(* PLC project OOP_Curso, Beckhoff Automation GmbH TwinCAT PLC Control 3.5.13.21 *)
(* stored: creationDateTime 2023-04-24T11:18:57.3670637, modificationDateTime 2023-04-24T11:18:57.3670637 *)

PROGRAM _12_Concepto_Keyword_Abstract
VAR
// 	fbLoadCell:REFERENCE TO AbstractLoadCell;
	
	ConcreteCSVLogger:ConcreteCSVLogger;
    ConcreteAdsLogger:ConcreteADSLogger;
    AbstractLogger:POINTER TO AbstractLogger;
    LogNow:BOOL;
    Process1:INT;
    Process2:INT;
END_VAR

            (*
Concepto ABSTRACTO
La palabra clave ABSTRACT está disponible para bloques de funciones, métodos y propiedades. Permite la implementación de un proyecto PLC con niveles de abstracción.
La abstracción es un concepto clave de la programación orientada a objetos. Los diferentes niveles de abstracción contienen aspectos de implementación generales o específicos.

CONCEPTO ABSTRACTO 1:	
Disponible en TC3.1 Build 4024

Aplicación de la abstracción
Es útil implementar funciones básicas o puntos en común de diferentes clases en una clase básica abstracta. Se implementan aspectos específicos en subclases no abstractas.
El principio es similar al uso de una interfaz. Las interfaces corresponden a clases puramente abstractas que contienen sólo métodos y propiedades abstractas.
Una clase abstracta también puede contener métodos y propiedades no abstractos.

Reglas para el uso de la palabra clave ABSTRACT
Los bloques de funciones abstractas no se pueden instanciar.
Los bloques de funciones abstractas pueden contener métodos y propiedades abstractos y no abstractos.
Los métodos abstractos o las propiedades no contienen ninguna implementación (solo la declaración).
Si un bloque de funciones contiene un método o propiedad abstracta, debe ser abstracta.
Los bloques de funciones abstractas deben extenderse para poder implementar los métodos o propiedades abstractas.
Por lo tanto: Un FB derivado debe implementar los métodos / propiedades de su FB básico o también debe definirse como abstracto.
Muestra
Clase básica abstracta:

FUNCTION_BLOCK ABSTRACT FB_System_Base
Los puntos en común de todos los módulos del sistema se implementan en esta clase básica abstracta. Contiene la propiedad no abstracta "nSystemID" y el método abstracto "Execute" para esto:

PROPERTY nSystemID : UINT
METHOD ABSTRACT Execute
mientras que la implementación de "nSystemID" es la misma para todos los sistemas, la implementación del método "Execute" difiere para los sistemas individuales.

Subclase no abstracta:

FUNCTION_BLOCK FB_StackSystem EXTENDS FB_System_Base
Las clases no abstractas que se derivan de la clase básica se implementan para los sistemas específicos. Esta subclase representa una pila. Dado que no es abstracto, debe implementar el método "Execute" que define la ejecución específica de la pila:

METHOD Execute

*)

// Process 1 assigns a logger and starts task 2.
CASE Process1 OF
    0: IF LogNow THEN
            LogNow:=FALSE;
            AbstractLogger:= ADR(ConcreteAdsLogger);
            Process2 :=1;
            Process1:=Process1+1;               
        END_IF
     
    1: IF Process2 = 0 THEN
            AbstractLogger:= ADR(ConcreteCSVLogger);
            Process2:=1;
            Process1:=Process1+1;   
       END_IF
        
     2:IF Process2 = 0 THEN
            AbstractLogger:= ADR(ConcreteAdsLogger);
            Process2:=1;
            Process1:=Process1+1;   
       END_IF
        
      3: IF Process2 = 0 THEN
            AbstractLogger:= ADR(ConcreteCSVLogger);
            Process2:=1;
            Process1:=Process1+1;   
       END_IF
        
      4:IF Process2 = 0 THEN
            Process1:=0;    
       END_IF
END_CASE
 
//Process 2 does its task indepently of the assigned type of logger. 
CASE process2 OF
    1: AbstractLogger^.LogMessage(CONCAT('Important message ',INT_TO_STRING(Process1)));
       process2:=process2+1;                
         
    2: AbstractLogger^();
       IF NOT AbstractLogger^.Busy THEN
            process2:=0;    
       END_IF
END_CASE
          
END_PROGRAM

FUNCTION_BLOCK ABSTRACT AbstractLoadCell
VAR_INPUT
END_VAR
VAR_OUTPUT
END_VAR
VAR
END_VAR

            
          

METHOD PUBLIC ABSTRACT GetActualValue : LREAL
VAR_INPUT
END_VAR
                  
                
END_METHOD
END_FUNCTION_BLOCK

FUNCTION_BLOCK ABSTRACT AbstractLogger

VAR
	_Busy:BOOL; //Backing variable for Busy property.
END_VAR

            
          

METHOD PROTECTED ABSTRACT InternalLog
VAR_INPUT
	Message:STRING;
END_VAR
                  
                
END_METHOD

METHOD PUBLIC LogMessage
VAR_INPUT
	Message:STRING;
END_VAR
VAR
    GetSystemTime : NT_GetTime:=(NetID:=''); //'xxx.xxx.xxx.1.1.1');
END_VAR
                  // Retrieve a the current system time and combine it with the input message. 
GetSystemTime(START:=FALSE);
REPEAT
    GetSystemTime(START:=TRUE);
UNTIL (NOT GetSystemTime.BUSY)
END_REPEAT
 
//Call abstract method
InternalLog(Message:=CONCAT(CONCAT(Message,', '),SYSTEMTIME_TO_STRING(GetSystemTime.TIMESTR)));
                
END_METHOD

{attribute 'monitoring' := 'variable'}
PROPERTY Busy : BOOL
GET
VAR
END_VAR
                    Busy:=_Busy;
                  
END_GET
SET
VAR
END_VAR
                    
                  
END_SET
END_PROPERTY
END_FUNCTION_BLOCK

FUNCTION_BLOCK PUBLIC FINAL ConcreteADSLogger EXTENDS AbstractLogger
VAR_INPUT
END_VAR
VAR_OUTPUT
END_VAR
VAR
END_VAR

            
          

METHOD PROTECTED InternalLog
VAR_INPUT
     Message:STRING;
END_VAR
                  _Busy:=TRUE;
 
ADSLOGSTR(    msgCtrlMask:=ADSLOG_MSGTYPE_LOG,
              msgFmtStr:=Message,
              strArg:='');
             
_Busy:=FALSE;
                
END_METHOD
END_FUNCTION_BLOCK

{attribute 'hide_all_locals'}
FUNCTION_BLOCK FINAL ConcreteCSVLogger EXTENDS AbstractLogger
VAR
    fbFileOpen:FB_FileOpen;
    fbFilePuts:FB_FilePuts;
    fbFileClose:FB_FileClose;
    State:INT;
    Message:STRING;
END_VAR

            CASE State OF
    0:  IF _Busy THEN
            State:=State+1;
        END_IF
     
    1:  fbFileOpen(bExecute:=FALSE);
        fbFileOpen(sNetId:='', //'xxx.xx.xxx.1.1.1',
            sPathName:='C:\Log.csv',
            nMode:=FOPEN_MODEAPPEND,
            bExecute:=TRUE);
        State:=State+1;
         
    2:  fbFileOpen(bExecute:=FALSE);
        IF NOT fbFileOpen.bBusy THEN
            State:=State+1;
        END_IF
     
    3:  fbFilePuts(bExecute :=FALSE);
        fbFilePuts( bExecute:=TRUE,
                    sNetId:='',//'xxx.xx.xxx.1.1.1',
                    hFile:=fbFileOpen.hFile,
                    sLine:=Message);
        State:=State+1;
     
    4:  fbFilePuts(bExecute:=FALSE);
        IF NOT fbFilePuts.bBusy THEN
            State:=State+1;
        END_IF
         
    5:  fbFileClose(bExecute :=FALSE);
        fbFileClose(sNetId:='',//'xxx.xx.xxx.1.1.1',
                    bExecute:=TRUE,
                    hFile:= fbFileOpen.hFile);
        State:=State+1; 
         
    6:  fbFileClose(bExecute:=FALSE);
        IF NOT fbFileClose.bBusy THEN
            State:=0;
            _Busy:=FALSE;
        END_IF
END_CASE       
          

METHOD PROTECTED  InternalLog
VAR_INPUT
    Message:STRING;
END_VAR
                  THIS^.Message:=CONCAT(Message,'$n');
_Busy:=TRUE;
                
END_METHOD
END_FUNCTION_BLOCK

FUNCTION_BLOCK PUBLIC ConcreteLoadCell EXTENDS AbstractLoadCell
VAR_INPUT
END_VAR
VAR_OUTPUT
END_VAR
VAR
END_VAR

            
          
END_FUNCTION_BLOCK
